Universal Robots PolyScope program: MainSimulation.urp

Program MainSimulation (createdIn=3.0.0 lastSavedIn=3.0.0 directory=. installation=default)
Robot Program (runOnlyOnce=true motionType=MoveJ speed=1.047198 acceleration=1.396263 useActiveTCP=false)
  Script file MainSimulation.script
    | def MainSimulation():
    |   # Global parameters:
    |   global speed_ms    = 0.250
    |   global speed_rads  = 0.750
    |   global accel_mss   = 1.200
    |   global accel_radss = 1.200
    |   global blend_radius_m = 0.001
    |   global ref_frame = p[0,0,0,0,0,0]
    | 
    |   #
    |   # TO REMOVE HEADER:
    |   # Go to "Program" -> "Post-Processor Editor"
    |   # Select "Universal Robots"
    |   # Set "INCLUDE_HEADER" to "False"
    |   #
    |   #--------------------------
    |   # Add any default subprograms here
    |   # For example, to drive a gripper as a program call:
    |   # def Gripper_Open():
    |   #   ...
    |   # end
    |   #
    |   # Example to drive a spray gun:
    |   def SprayOn(value):
    |     # use the value as an output:
    |     DO_SPRAY = 5
    |     if value == 0:
    |       set_standard_digital_out(DO_SPRAY, False)
    |     else:
    |       set_standard_digital_out(DO_SPRAY, True)
    |     end
    |   end
    | 
    |   # Example to drive an extruder:
    |   def Extruder(value):
    |     # use the value as an output:
    |     if value < 0:
    |       # stop extruder
    |     else:
    |       # start extruder
    |     end
    |   end
    | 
    |   # Example to move an external axis
    |   def MoveAxis(value):
    |     # use the value as an output:
    |     DO_AXIS_1 = 1
    |     DI_AXIS_1 = 1
    |     if value <= 0:
    |       set_standard_digital_out(DO_AXIS_1, False)
    | 
    |       # Wait for digital input to change state
    |       #while (get_standard_digital_in(DI_AXIS_1) != False):
    |       #  sync()
    |       #end
    |     else:
    |       set_standard_digital_out(DO_AXIS_1, True)
    | 
    |       # Wait for digital input to change state
    |       #while (get_standard_digital_in(DI_AXIS_1) != True):
    |       #  sync()
    |       #end
    |     end
    |   end
    |   #--------------------------
    | 
    | 
    |   # Main program:
    |   # Program generated by RoboDK v5.6.4 for UR10 A on 06/12/2023 15:10:39
    |   # Using nominal kinematics.
    |   PrepareSimulation()
    |   SimulateCamera()
    |   MoveConveyor
    |   PartsToConveyor
    |   PartsToPallet()
    |   # End of main program
    | end
    | 
    | MainSimulation()
